{attribute 'GeneratedUsingTerminal: EPP3744-0041-0016'}
{attribute addProperty BoxType "EPP3744-0041-0016"}
{attribute addProperty Id "DIG_InputsAT %I*DIG_Inputs_697E0EF26AI_Inputs_Channel_1AT %I*AI_Inputs_Channel_4521310411AI_Inputs_Channel_2AT %I*AI_Inputs_Channel_4521310411AI_Inputs_Channel_3AT %I*AI_Inputs_Channel_4521310411AI_Inputs_Channel_4AT %I*AI_Inputs_Channel_4521310411DEV_Inputs_DeviceAT %I*DEV_Inputs_Device_5F4E175E5DIG_OutputsAT %Q*DIG_Outputs_DE230DD52DEV_Outputs_DeviceAT %Q*DEV_Outputs_Device_59FFD2471WcStateAT %I*WcState_9091E0EB2InfoDataAT %I*InfoData_32EB74EA10"}
{attribute addProperty CRC "828150484"}
{attribute addProperty Size "70"}
TYPE EPP3744_315C92D4 EXTENDS EtcSlaveTerminalBase_947E5A46 :
STRUCT
	{attribute addProperty Name "DIG_Inputs"}
	DIG_Inputs : DIG_Inputs_697E0EF2;
	{attribute addProperty Name "AI_Inputs_Channel_1"}
	AI_Inputs_Channel_1 : AI_Inputs_Channel_45213104;
	{attribute addProperty Name "AI_Inputs_Channel_2"}
	AI_Inputs_Channel_2 : AI_Inputs_Channel_45213104;
	{attribute addProperty Name "AI_Inputs_Channel_3"}
	AI_Inputs_Channel_3 : AI_Inputs_Channel_45213104;
	{attribute addProperty Name "AI_Inputs_Channel_4"}
	AI_Inputs_Channel_4 : AI_Inputs_Channel_45213104;
	{attribute addProperty Name "DEV_Inputs_Device"}
	DEV_Inputs_Device : DEV_Inputs_Device_5F4E175E;
	{attribute addProperty Name "DIG_Outputs"}
	DIG_Outputs : DIG_Outputs_DE230DD5;
	{attribute addProperty Name "DEV_Outputs_Device"}
	DEV_Outputs_Device : DEV_Outputs_Device_59FFD247;
	{attribute addProperty Name "WcState"}
	WcState : WcState_9091E0EB;
	{attribute addProperty Name "InfoData"}
	InfoData : InfoData_32EB74EA;
END_STRUCT
END_TYPE

(* stored: Version 1.2.0.0, ProductVersion 3.1.4024.9
   DUT EPP3744_315C92D4: Id {7bb7c161-e369-4b7c-90ff-a6b870bc78db} *)
